Staubli VAL3: loadType.pgx

program loadType(num& x_nResult[])
  local num i
  local num l_nIndex
  local string l_sPath
begin
  if find(trajType:libPath(),saveData:sTrajTypeUsing)==-1
    // load the traj type
    call saveData:getPathInstr(saveData:sTrajTypeUsing,l_sPath)
    x_nResult=trajType:libLoad(l_sPath)
    delay(0)
    if x_nResult!=0
      popUpMsg("error load traj type on START "+saveData:sTrajTypeUsing+toString("",x_nResult))
    endIf
  endIf
end
